// TIA Portal V19 export
FUNCTION "FC50_RecipeManage" : Void   // FC50, LAD
{ S7_Optimized_Access := 'TRUE' }
// stored: AutoNumber false, IsIECCheckEnabled true, SetENOAutomatically false
BEGIN

REGION Network 1: Management of recipde (Load, Save, Creat )
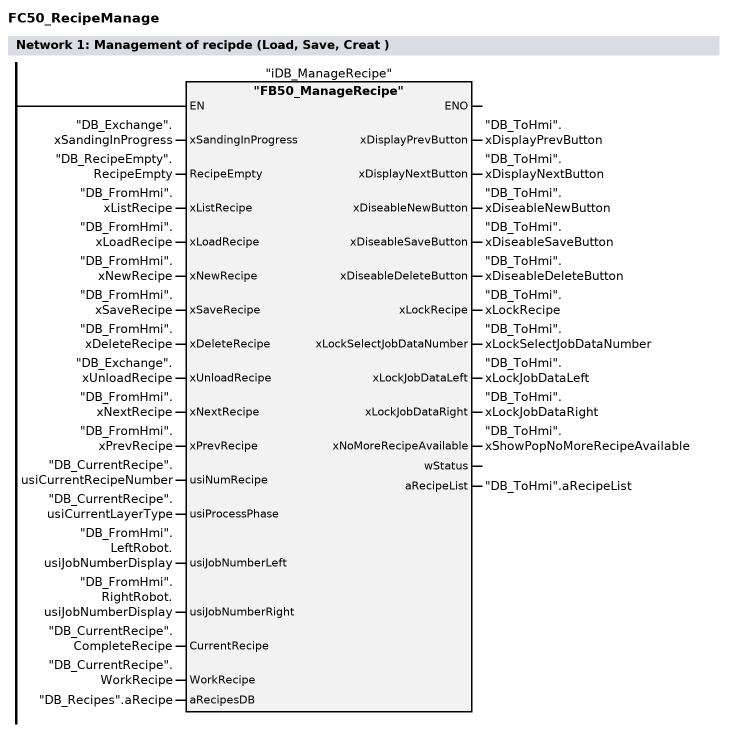
   RUNG wire#powerrail
      "iDB_ManageRecipe"(xSandingInProgress := "DB_Exchange".xSandingInProgress, RecipeEmpty := "DB_RecipeEmpty".RecipeEmpty, xListRecipe := "DB_FromHmi".xListRecipe, xLoadRecipe := "DB_FromHmi".xLoadRecipe, xNewRecipe := "DB_FromHmi".xNewRecipe, xSaveRecipe := "DB_FromHmi".xSaveRecipe, xDeleteRecipe := "DB_FromHmi".xDeleteRecipe, xUnloadRecipe := "DB_Exchange".xUnloadRecipe, xNextRecipe := "DB_FromHmi".xNextRecipe, xPrevRecipe := "DB_FromHmi".xPrevRecipe, usiNumRecipe := "DB_CurrentRecipe".usiCurrentRecipeNumber, usiProcessPhase := "DB_CurrentRecipe".usiCurrentLayerType, usiJobNumberLeft := "DB_FromHmi".LeftRobot.usiJobNumberDisplay, usiJobNumberRight := "DB_FromHmi".RightRobot.usiJobNumberDisplay, CurrentRecipe := "DB_CurrentRecipe".CompleteRecipe, WorkRecipe := "DB_CurrentRecipe".WorkRecipe, aRecipesDB := "DB_Recipes".aRecipe, xDisplayPrevButton => "DB_ToHmi".xDisplayPrevButton, xDisplayNextButton => "DB_ToHmi".xDisplayNextButton, xDiseableNewButton => "DB_ToHmi".xDiseableNewButton, xDiseableSaveButton => "DB_ToHmi".xDiseableSaveButton, xDiseableDeleteButton => "DB_ToHmi".xDiseableDeleteButton, xLockRecipe => "DB_ToHmi".xLockRecipe, xLockSelectJobDataNumber => "DB_ToHmi".xLockSelectJobDataNumber, xLockJobDataLeft => "DB_ToHmi".xLockJobDataLeft, xLockJobDataRight => "DB_ToHmi".xLockJobDataRight, xNoMoreRecipeAvailable => "DB_ToHmi".xShowPopNoMoreRecipeAvailable, wStatus =>, aRecipeList => "DB_ToHmi".aRecipeList)
   END_RUNG
   // the same network as SCL:
   "iDB_ManageRecipe"(xSandingInProgress := "DB_Exchange".xSandingInProgress,   // "FB50_ManageRecipe"
                      RecipeEmpty := "DB_RecipeEmpty".RecipeEmpty,
                      xListRecipe := "DB_FromHmi".xListRecipe,
                      xLoadRecipe := "DB_FromHmi".xLoadRecipe,
                      xNewRecipe := "DB_FromHmi".xNewRecipe,
                      xSaveRecipe := "DB_FromHmi".xSaveRecipe,
                      xDeleteRecipe := "DB_FromHmi".xDeleteRecipe,
                      xUnloadRecipe := "DB_Exchange".xUnloadRecipe,
                      xNextRecipe := "DB_FromHmi".xNextRecipe,
                      xPrevRecipe := "DB_FromHmi".xPrevRecipe,
                      usiNumRecipe := "DB_CurrentRecipe".usiCurrentRecipeNumber,
                      usiProcessPhase := "DB_CurrentRecipe".usiCurrentLayerType,
                      usiJobNumberLeft := "DB_FromHmi".LeftRobot.usiJobNumberDisplay,
                      usiJobNumberRight := "DB_FromHmi".RightRobot.usiJobNumberDisplay,
                      CurrentRecipe := "DB_CurrentRecipe".CompleteRecipe,
                      WorkRecipe := "DB_CurrentRecipe".WorkRecipe,
                      aRecipesDB := "DB_Recipes".aRecipe,
                      xDisplayPrevButton => "DB_ToHmi".xDisplayPrevButton,
                      xDisplayNextButton => "DB_ToHmi".xDisplayNextButton,
                      xDiseableNewButton => "DB_ToHmi".xDiseableNewButton,
                      xDiseableSaveButton => "DB_ToHmi".xDiseableSaveButton,
                      xDiseableDeleteButton => "DB_ToHmi".xDiseableDeleteButton,
                      xLockRecipe => "DB_ToHmi".xLockRecipe,
                      xLockSelectJobDataNumber => "DB_ToHmi".xLockSelectJobDataNumber,
                      xLockJobDataLeft => "DB_ToHmi".xLockJobDataLeft,
                      xLockJobDataRight => "DB_ToHmi".xLockJobDataRight,
                      xNoMoreRecipeAvailable => "DB_ToHmi".xShowPopNoMoreRecipeAvailable,
                      aRecipeList => "DB_ToHmi".aRecipeList);
END_REGION
END_FUNCTION
